FUNCTION_BLOCK MOD_Occupation (* Module occupation: OPC UA methods Occupy(Session) and Release(Session) answer [Accepted, ErrorID]; publishes Occupied (never the session ID) and shares the owner on a local channel *)
  (* Standard: 61499-2 *)
  (* Version 0.1, 2026-09-28, Project contributors, AAU Smart Production Lab *)
  PACKAGE modlib;
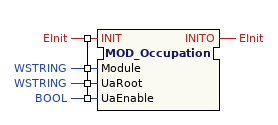
  EVENT_INPUT
    INIT : EInit WITH Module, UaRoot, UaEnable;
  END_EVENT
  EVENT_OUTPUT
    INITO : EInit;
  END_EVENT
  VAR_INPUT
    Module : WSTRING;
    UaRoot : WSTRING;
    UaEnable : BOOL;
  END_VAR
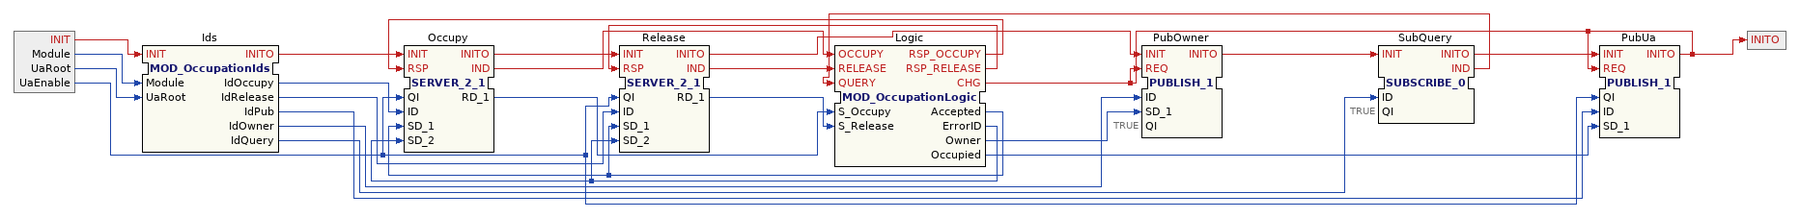
  FBS
    Ids : modlib::MOD_OccupationIds;
    Occupy : iec61499::net::SERVER_2_1;
    Release : iec61499::net::SERVER_2_1;
    Logic : modlib::MOD_OccupationLogic;
    PubOwner : iec61499::net::PUBLISH_1(QI := TRUE);
    SubQuery : iec61499::net::SUBSCRIBE_0(QI := TRUE);
    PubUa : iec61499::net::PUBLISH_1;
  END_FBS
  EVENT_CONNECTIONS
    INIT TO Ids.INIT;
    Ids.INITO TO Occupy.INIT;
    Occupy.INITO TO Release.INIT;
    Release.INITO TO PubOwner.INIT;
    PubOwner.INITO TO SubQuery.INIT;
    SubQuery.INITO TO PubUa.INIT;
    PubUa.INITO TO PubUa.REQ;
    PubUa.INITO TO INITO;
    Occupy.IND TO Logic.OCCUPY;
    Logic.RSP_OCCUPY TO Occupy.RSP;
    Release.IND TO Logic.RELEASE;
    Logic.RSP_RELEASE TO Release.RSP;
    SubQuery.IND TO Logic.QUERY;
    Logic.CHG TO PubOwner.REQ;
    Logic.CHG TO PubUa.REQ;
  END_CONNECTIONS
  DATA_CONNECTIONS
    Module TO Ids.Module;
    UaRoot TO Ids.UaRoot;
    UaEnable TO Occupy.QI;
    UaEnable TO Release.QI;
    UaEnable TO PubUa.QI;
    Ids.IdOccupy TO Occupy.ID;
    Ids.IdRelease TO Release.ID;
    Ids.IdPub TO PubUa.ID;
    Ids.IdOwner TO PubOwner.ID;
    Ids.IdQuery TO SubQuery.ID;
    Occupy.RD_1 TO Logic.S_Occupy;
    Logic.Accepted TO Occupy.SD_1;
    Logic.ErrorID TO Occupy.SD_2;
    Release.RD_1 TO Logic.S_Release;
    Logic.Accepted TO Release.SD_1;
    Logic.ErrorID TO Release.SD_2;
    Logic.Owner TO PubOwner.SD_1;
    Logic.Occupied TO PubUa.SD_1;
  END_CONNECTIONS
END_FUNCTION_BLOCK
